TYPE AssemblyComRequest :
STRUCT
  Start : BOOL;
  Stop : BOOL;
  GoHome : BOOL;
  Halt : BOOL;
END_STRUCT
END_TYPE

(* stored: Version 1.1.0.1
   DUT AssemblyComRequest: Id {f05e98db-850b-4817-8a45-a28700d114ca} *)
